// TIA Portal project "IndustrialSortingAutomation" (V17)
// Vorlageprojekt für das Buch mit Zielsystem S7-1200

(* hardware
DEVICE "S7-1200-Station_1"  S7-1200 Station
   slot 0: "Baugruppenträger_0"  Rack  V1.0
   slot 1: "PLC_1"  CPU 1211C DC/DC/DC  6ES7 211-1AE40-0XB0  V4.1
DEVICE "HMI_1"  KTP900 Basic PN
   slot 0: "HMI_1"  KTP900 Basic PN  6AV2 123-2JB03-0AX0  17.0.0.0
   slot 1: "HMI_RT_1"  KTP900 Basic PN  6AV2 123-2JB03-0AX0  17.0.0.0
   slot 5: "HMI_1.IE_CP_1"  PROFINET Interface  17.0.0.0
      slot 1: "PROFINET Interface_1"  PROFINET Interface
         slot 1: "Port_1"  Port
*)

// ===== PLC "PLC_1"  CPU 1211C DC/DC/DC =====

VAR_GLOBAL   // PLC tag table "Standard-Variablentabelle"
   "Motore_P" AT %A0.0 : Bool;
   "Sensore_P" AT %E0.0 : Bool;
   "Sensore_R" AT %E0.1 : Bool;
   "System_Byte" AT %MB1 : Byte;
   "FirstScan" AT %M1.0 : Bool;
   "DiagStatusUpdate" AT %M1.1 : Bool;
   "AlwaysTRUE" AT %M1.2 : Bool;
   "AlwaysFALSE" AT %M1.3 : Bool;
   "M_Pronto_P" AT %M10.0 : Bool;
   "M_Pronto_R" AT %M10.1 : Bool;
   "M_VAI_P" AT %M10.2 : Bool;
   "M_VAI_R" AT %M10.3 : Bool;
   "Cont_B_Board" AT %QW30 : Int;
   "Cont_V_Board" AT %QW32 : Int;
   "Cont_G_Board" AT %QW34 : Int;
   "Cont_P_Board" AT %QW36 : Int;
   "Motore_R" AT %Q0.1 : Bool;
   "Sorter_Pacchi_Turn" AT %Q0.2 : Bool;
   "Sorter_Pacchi_Belt" AT %Q0.3 : Bool;
   "Motore_Nastro_Ingresso_Smistamento" AT %Q0.4 : Bool;
   "Sorter_Raw_Blu_Turn" AT %Q0.5 : Bool;
   "Sorter_Raw_Blu_Belt" AT %Q0.6 : Bool;
   "Sorter_Raw_Verde_Turn" AT %Q0.7 : Bool;
   "Sorter_Raw_Verde_Belt" AT %Q1.0 : Bool;
   "Sorter_Raw_Grigio_Turn" AT %Q1.1 : Bool;
   "Sorter_Raw_Grigio_Belt" AT %Q1.2 : Bool;
   "Motore_Nastro_Comune" AT %Q2.0 : Bool;
   "Motore_Nastro_Uscita_P" AT %Q2.1 : Bool;
   "Motore_Nastro_Uscita_R" AT %Q2.2 : Bool;
   "Motore_Nastro_Smistamento" AT %Q2.3 : Bool;
   "Motore_Nastro_Uscita_B" AT %Q2.4 : Bool;
   "Motore_Nastro_Uscita_V" AT %Q2.5 : Bool;
   "Motore_Nastro_Uscita_G" AT %Q2.6 : Bool;
   "Sensore_Deviatore__P" AT %I0.2 : Bool;
   "Sensore_Uscita_P" AT %I0.3 : Bool;
   "Sensore_Uscita_R" AT %I0.4 : Bool;
   "Sensore_Fine_Incrocio" AT %I0.5 : Bool;
   "M_Apri_Grigio" AT %M2.2 : Bool;
   "M_AVA_Smistamento" AT %M2.3 : Bool;
   "M_Apri_Blu" AT %M2.0 : Bool;
   "M_Apri_Verde" AT %M2.1 : Bool;
   "Vision_Sensor" AT %IW30 : Int;
   "Cont_B" AT %MW100 : Int;
   "Cont_V" AT %MW102 : Int;
   "Cont_G" AT %MW104 : Int;
   "Cont_P" AT %MW106 : Int;
   "Emergency_Stop" AT %I0.6 : Bool;
   "Waring_Light" AT %Q1.3 : Bool;
   "M_Motore_P" AT %M3.0 : Bool;
   "M_Motore_R" AT %M3.1 : Bool;
   "M_Turn_P" AT %M3.2 : Bool;
   "M_Belt_P" AT %M3.3 : Bool;
   "M_Turn_B" AT %M3.4 : Bool;
   "M_Belt_B" AT %M3.5 : Bool;
   "M_Turn_V" AT %M3.6 : Bool;
   "M_Belt_V" AT %M3.7 : Bool;
   "M_Turn_G" AT %M4.0 : Bool;
   "M_Belt_G" AT %M4.1 : Bool;
   "Alarm_Siren" AT %Q1.4 : Bool;
END_VAR

DATA_BLOCK "FB_Nastro_Ingresso_DB_Pacchi"   // DB1
{ S7_Optimized_Access := 'TRUE' }
VERSION : 0.1
// stored: InstanceOfName FB_Nastro_Ingresso
"FB_Nastro_Ingresso"
BEGIN
END_DATA_BLOCK

DATA_BLOCK "FB_Nastro_Ingresso_DB_Raw"   // DB2
{ S7_Optimized_Access := 'TRUE' }
VERSION : 0.1
// stored: InstanceOfName FB_Nastro_Ingresso
"FB_Nastro_Ingresso"
BEGIN
END_DATA_BLOCK

DATA_BLOCK "FB_Gestore_Incrocio_DB"   // DB3
{ S7_Optimized_Access := 'TRUE' }
VERSION : 0.1
// stored: InstanceOfName FB_Gestore_Incrocio
"FB_Gestore_Incrocio"
BEGIN
END_DATA_BLOCK

DATA_BLOCK "FB_Deviatore_DB_Pacchi"   // DB4
{ S7_Optimized_Access := 'TRUE' }
VERSION : 0.1
// stored: InstanceOfName FB_Deviatore
"FB_Deviatore"
BEGIN
END_DATA_BLOCK

DATA_BLOCK "FB_Gestore_Smistamento_DB"   // DB5
{ S7_Optimized_Access := 'TRUE' }
VERSION : 0.1
// stored: InstanceOfName FB_Gestore_Smistamento
"FB_Gestore_Smistamento"
BEGIN
END_DATA_BLOCK

DATA_BLOCK "FB_Deviatore_DB_Blu"   // DB6
{ S7_Optimized_Access := 'TRUE' }
VERSION : 0.1
// stored: InstanceOfName FB_Deviatore
"FB_Deviatore"
BEGIN
END_DATA_BLOCK

DATA_BLOCK "FB_Deviatore_DB_Verde"   // DB7
{ S7_Optimized_Access := 'TRUE' }
VERSION : 0.1
// stored: InstanceOfName FB_Deviatore
"FB_Deviatore"
BEGIN
END_DATA_BLOCK

DATA_BLOCK "FB_Deviatore_DB_Grigio"   // DB8
{ S7_Optimized_Access := 'TRUE' }
VERSION : 0.1
// stored: InstanceOfName FB_Deviatore
"FB_Deviatore"
BEGIN
END_DATA_BLOCK

// folder: System blocks/Program resources

DATA_BLOCK "IEC_Timer_0_DB_Nastro_Smistamento"   // DB9
{ S7_Optimized_Access := 'TRUE' }
AUTHOR : Simatic
FAMILY : IEC
NAME : IEC_TMR
VERSION : 1.0
// stored: InstanceOfName IEC_TIMER
"IEC_TIMER"
BEGIN
END_DATA_BLOCK

// folder: (top level)

FUNCTION_BLOCK "FB_Nastro_Ingresso"   // FB1, LAD
{ S7_Optimized_Access := 'TRUE' }
VERSION : 0.1
   VAR_INPUT
      fn : Bool;
      VAI : Bool;
      Tempo_Spinta : Time;
   END_VAR
   VAR_OUTPUT
      AVA : Bool;
      pronto : Bool;
   END_VAR
   VAR
      f0 : Bool;
      f1 : Bool;
      f2 : Bool;
      f3 : Bool;
      tr1 : Bool;
      tr2 : Bool;
      tr3 : Bool;
      tr4 : Bool;
      Timer_Attr : IEC_TIMER;
   END_VAR
BEGIN

REGION Network 1: Inizializzazione
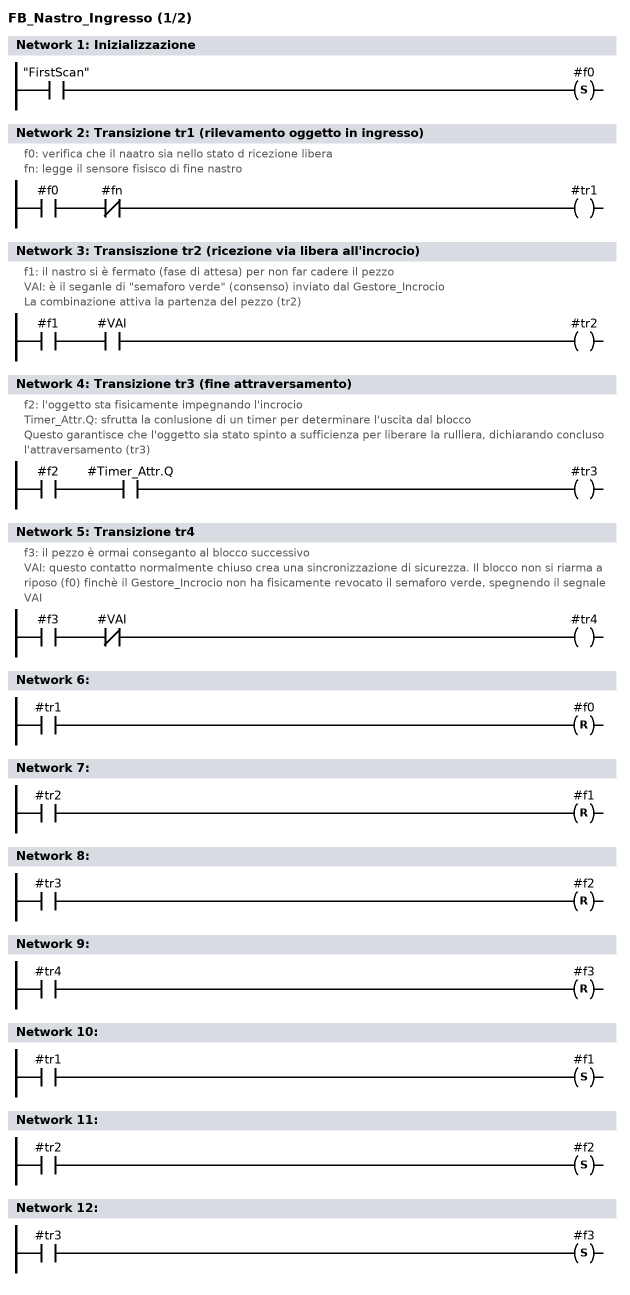
   RUNG wire#powerrail
      Contact( "FirstScan" )
      S_Coil( #f0 )
   END_RUNG
   // the same network as SCL:
   IF "FirstScan" THEN #f0 := TRUE; END_IF;
END_REGION

REGION Network 2: Transizione tr1 (rilevamento oggetto in ingresso)
   // f0: verifica che il naatro sia nello stato d ricezione libera
   // fn: legge il sensore fisisco di fine nastro
   RUNG wire#powerrail
      Contact( #f0 )
      I_Contact( #fn )
      Coil( #tr1 )
   END_RUNG
   // the same network as SCL:
   #tr1 := #f0 AND NOT #fn;
END_REGION

REGION Network 3: Transiszione tr2 (ricezione via libera all'incrocio)
   // f1: il nastro si è fermato (fase di attesa) per non far cadere il pezzo
   // VAI: è il seganle di "semaforo verde" (consenso) inviato dal Gestore_Incrocio
   // La combinazione attiva la partenza del pezzo (tr2)
   RUNG wire#powerrail
      Contact( #f1 )
      Contact( #VAI )
      Coil( #tr2 )
   END_RUNG
   // the same network as SCL:
   #tr2 := #f1 AND #VAI;
END_REGION

REGION Network 4: Transizione tr3 (fine attraversamento)
   // f2: l'oggetto sta fisicamente impegnando l'incrocio
   // Timer_Attr.Q: sfrutta la conlusione di un timer per determinare l'uscita dal blocco
   // Questo garantisce che l'oggetto sia stato spinto a sufficienza per liberare la rulliera, dichiarando concluso l'attraversamento (tr3)
   RUNG wire#powerrail
      Contact( #f2 )
      Contact( #Timer_Attr.Q )
      Coil( #tr3 )
   END_RUNG
   // the same network as SCL:
   #tr3 := #f2 AND #Timer_Attr.Q;
END_REGION

REGION Network 5: Transizione tr4
   // f3: il pezzo è ormai conseganto al blocco successivo 
   // VAI: questo contatto normalmente chiuso crea una sincronizzazione di sicurezza. Il blocco non si riarma a riposo (f0) finchè il Gestore_Incrocio non ha fisicamente revocato il semaforo verde, spegnendo il segnale VAI
   RUNG wire#powerrail
      Contact( #f3 )
      I_Contact( #VAI )
      Coil( #tr4 )
   END_RUNG
   // the same network as SCL:
   #tr4 := #f3 AND NOT #VAI;
END_REGION

REGION Network 6
   RUNG wire#powerrail
      Contact( #tr1 )
      R_Coil( #f0 )
   END_RUNG
   // the same network as SCL:
   IF #tr1 THEN #f0 := FALSE; END_IF;
END_REGION

REGION Network 7
   RUNG wire#powerrail
      Contact( #tr2 )
      R_Coil( #f1 )
   END_RUNG
   // the same network as SCL:
   IF #tr2 THEN #f1 := FALSE; END_IF;
END_REGION

REGION Network 8
   RUNG wire#powerrail
      Contact( #tr3 )
      R_Coil( #f2 )
   END_RUNG
   // the same network as SCL:
   IF #tr3 THEN #f2 := FALSE; END_IF;
END_REGION

REGION Network 9
   RUNG wire#powerrail
      Contact( #tr4 )
      R_Coil( #f3 )
   END_RUNG
   // the same network as SCL:
   IF #tr4 THEN #f3 := FALSE; END_IF;
END_REGION

REGION Network 10
   RUNG wire#powerrail
      Contact( #tr1 )
      S_Coil( #f1 )
   END_RUNG
   // the same network as SCL:
   IF #tr1 THEN #f1 := TRUE; END_IF;
END_REGION

REGION Network 11
   RUNG wire#powerrail
      Contact( #tr2 )
      S_Coil( #f2 )
   END_RUNG
   // the same network as SCL:
   IF #tr2 THEN #f2 := TRUE; END_IF;
END_REGION

REGION Network 12
   RUNG wire#powerrail
      Contact( #tr3 )
      S_Coil( #f3 )
   END_RUNG
   // the same network as SCL:
   IF #tr3 THEN #f3 := TRUE; END_IF;
END_REGION

REGION Network 13
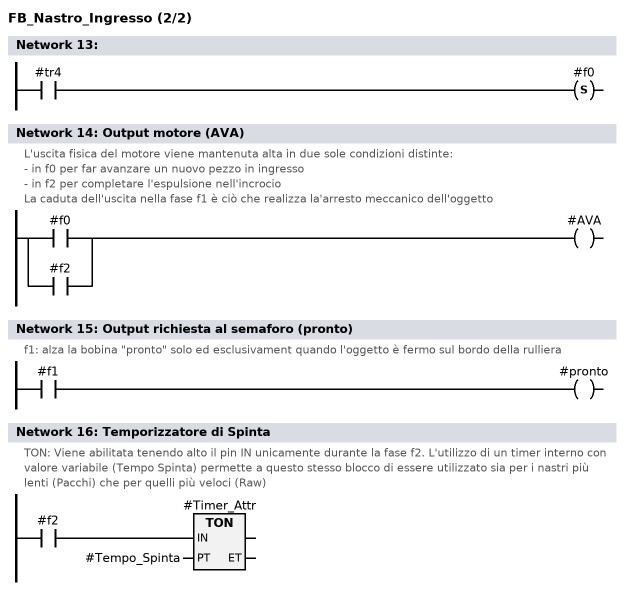
   RUNG wire#powerrail
      Contact( #tr4 )
      S_Coil( #f0 )
   END_RUNG
   // the same network as SCL:
   IF #tr4 THEN #f0 := TRUE; END_IF;
END_REGION

REGION Network 14: Output motore (AVA)
   // L'uscita fisica del motore viene mantenuta alta in due sole condizioni distinte:
   // - in f0 per far avanzare un nuovo pezzo in ingresso
   // - in f2 per completare l'espulsione nell'incrocio
   // La caduta dell'uscita nella fase f1 è ciò che realizza la'arresto meccanico dell'oggetto
   RUNG wire#powerrail
      Contact( #f0 )
      wire#w1
      Coil( #AVA )
   END_RUNG
   RUNG wire#powerrail
      Contact( #f2 )
   END_RUNG wire#w1
   // the same network as SCL:
   #AVA := #f0 OR #f2;
END_REGION

REGION Network 15: Output richiesta al semaforo (pronto)
   // f1: alza la bobina "pronto" solo ed esclusivament quando l'oggetto è fermo sul bordo della rulliera
   RUNG wire#powerrail
      Contact( #f1 )
      Coil( #pronto )
   END_RUNG
   // the same network as SCL:
   #pronto := #f1;
END_REGION

REGION Network 16: Temporizzatore di Spinta
   // TON: Viene abilitata tenendo alto il pin IN unicamente durante la fase f2. L'utilizzo di un timer interno con valore variabile (Tempo Spinta) permette a questo stesso blocco di essere utilizzato sia per i nastri più lenti (Pacchi) che per quelli più veloci (Raw)
   #Timer_Attr.TON(IN := #f2, PT := #Tempo_Spinta);
END_REGION
END_FUNCTION_BLOCK

FUNCTION_BLOCK "FB_Gestore_Incrocio"   // FB2, LAD
{ S7_Optimized_Access := 'TRUE' }
VERSION : 0.1
   VAR_INPUT
      pronto_P : Bool;
      pronto_R : Bool;
      Pass : Bool;
   END_VAR
   VAR_OUTPUT
      VAI_P : Bool;
      VAI_R : Bool;
   END_VAR
   VAR
      f0 : Bool;
      f1 : Bool;
      f2 : Bool;
      tr1 : Bool;
      tr2 : Bool;
      tr3 : Bool;
      tr4 : Bool;
      Mem_Fronte_P : Bool;
      Mem_Fronte_R : Bool;
   END_VAR
   VAR_TEMP   // added for the SCL form of the ladder/FBD networks
      _w1 : Bool;
   END_VAR
BEGIN

REGION Network 1: Inizializzazione
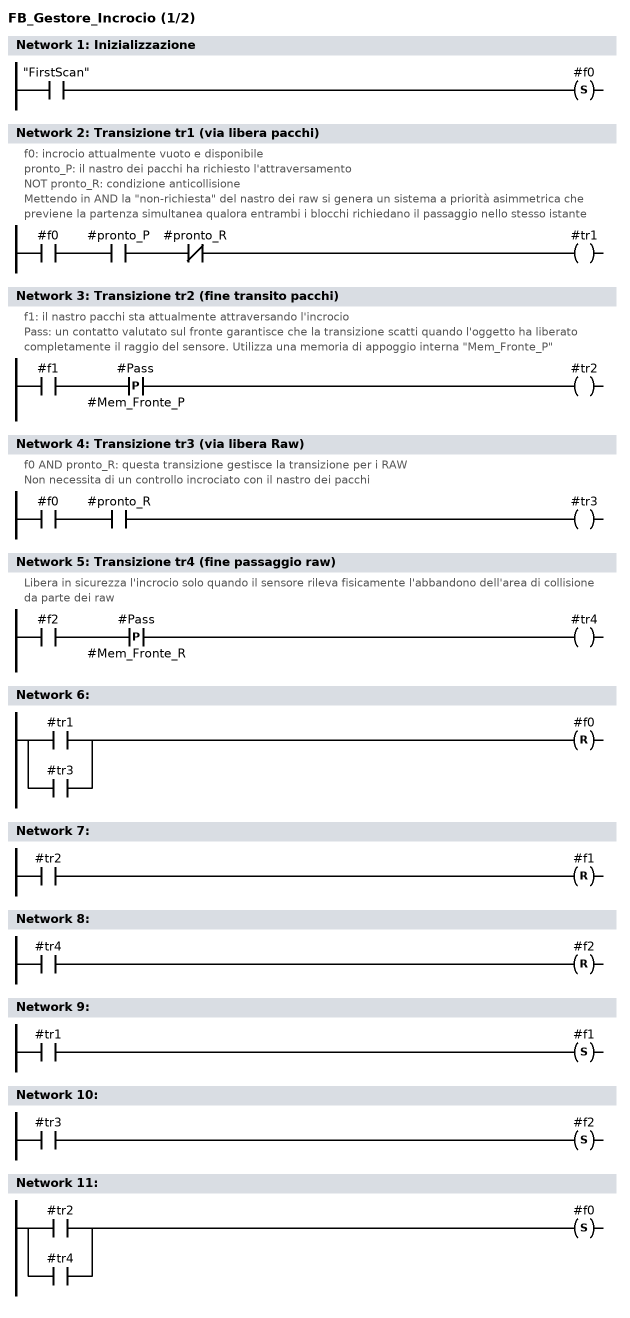
   RUNG wire#powerrail
      Contact( "FirstScan" )
      S_Coil( #f0 )
   END_RUNG
   // the same network as SCL:
   IF "FirstScan" THEN #f0 := TRUE; END_IF;
END_REGION

REGION Network 2: Transizione tr1 (via libera pacchi)
   // f0: incrocio attualmente vuoto e disponibile
   // pronto_P: il nastro dei pacchi ha richiesto l'attraversamento
   // NOT pronto_R: condizione anticollisione
   // Mettendo in AND la "non-richiesta" del nastro dei raw si genera un sistema a priorità asimmetrica che previene la partenza simultanea qualora entrambi i blocchi richiedano il passaggio nello stesso istante
   RUNG wire#powerrail
      Contact( #f0 )
      Contact( #pronto_P )
      I_Contact( #pronto_R )
      Coil( #tr1 )
   END_RUNG
   // the same network as SCL:
   #tr1 := #f0 AND #pronto_P AND NOT #pronto_R;
END_REGION

REGION Network 3: Transizione tr2 (fine transito pacchi)
   // f1: il nastro pacchi sta attualmente attraversando l'incrocio
   // Pass: un contatto valutato sul fronte garantisce che la transizione scatti quando l'oggetto ha liberato completamente il raggio del sensore. Utilizza una memoria di appoggio interna "Mem_Fronte_P"
   RUNG wire#powerrail
      Contact( #f1 )
      P_Contact(operand := #Pass, bit := #Mem_Fronte_P)
      Coil( #tr2 )
   END_RUNG
   // the same network as SCL:
   #_w1 := #f1 AND #Pass AND NOT #Mem_Fronte_P;   // rising edge of #Pass
   #Mem_Fronte_P := #Pass;
   #tr2 := #_w1;
END_REGION

REGION Network 4: Transizione tr3 (via libera Raw)
   // f0 AND pronto_R: questa transizione gestisce la transizione per i RAW
   // Non necessita di un controllo incrociato con il nastro dei pacchi
   RUNG wire#powerrail
      Contact( #f0 )
      Contact( #pronto_R )
      Coil( #tr3 )
   END_RUNG
   // the same network as SCL:
   #tr3 := #f0 AND #pronto_R;
END_REGION

REGION Network 5: Transizione tr4 (fine passaggio raw)
   // Libera in sicurezza l'incrocio solo quando il sensore rileva fisicamente l'abbandono dell'area di collisione da parte dei raw
   RUNG wire#powerrail
      Contact( #f2 )
      P_Contact(operand := #Pass, bit := #Mem_Fronte_R)
      Coil( #tr4 )
   END_RUNG
   // the same network as SCL:
   #_w1 := #f2 AND #Pass AND NOT #Mem_Fronte_R;   // rising edge of #Pass
   #Mem_Fronte_R := #Pass;
   #tr4 := #_w1;
END_REGION

REGION Network 6
   RUNG wire#powerrail
      Contact( #tr1 )
      wire#w1
      R_Coil( #f0 )
   END_RUNG
   RUNG wire#powerrail
      Contact( #tr3 )
   END_RUNG wire#w1
   // the same network as SCL:
   IF #tr1 OR #tr3 THEN #f0 := FALSE; END_IF;
END_REGION

REGION Network 7
   RUNG wire#powerrail
      Contact( #tr2 )
      R_Coil( #f1 )
   END_RUNG
   // the same network as SCL:
   IF #tr2 THEN #f1 := FALSE; END_IF;
END_REGION

REGION Network 8
   RUNG wire#powerrail
      Contact( #tr4 )
      R_Coil( #f2 )
   END_RUNG
   // the same network as SCL:
   IF #tr4 THEN #f2 := FALSE; END_IF;
END_REGION

REGION Network 9
   RUNG wire#powerrail
      Contact( #tr1 )
      S_Coil( #f1 )
   END_RUNG
   // the same network as SCL:
   IF #tr1 THEN #f1 := TRUE; END_IF;
END_REGION

REGION Network 10
   RUNG wire#powerrail
      Contact( #tr3 )
      S_Coil( #f2 )
   END_RUNG
   // the same network as SCL:
   IF #tr3 THEN #f2 := TRUE; END_IF;
END_REGION

REGION Network 11
   RUNG wire#powerrail
      Contact( #tr2 )
      wire#w1
      S_Coil( #f0 )
   END_RUNG
   RUNG wire#powerrail
      Contact( #tr4 )
   END_RUNG wire#w1
   // the same network as SCL:
   IF #tr2 OR #tr4 THEN #f0 := TRUE; END_IF;
END_REGION

REGION Network 12: Output consenso pacchi
   // VAI_P: il segnale di "semaforo verde" per la linea dei pacchi  viene pilotato dallo stato f1. Finchè f1 è ativo il permesso rimane alto generando il flusso continuo.
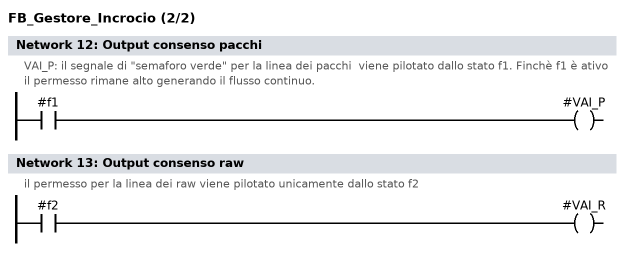
   RUNG wire#powerrail
      Contact( #f1 )
      Coil( #VAI_P )
   END_RUNG
   // the same network as SCL:
   #VAI_P := #f1;
END_REGION

REGION Network 13: Output consenso raw
   // il permesso per la linea dei raw viene pilotato unicamente dallo stato f2
   RUNG wire#powerrail
      Contact( #f2 )
      Coil( #VAI_R )
   END_RUNG
   // the same network as SCL:
   #VAI_R := #f2;
END_REGION
END_FUNCTION_BLOCK

FUNCTION_BLOCK "FB_Deviatore"   // FB3, LAD
{ S7_Optimized_Access := 'TRUE' }
VERSION : 0.1
   VAR_INPUT
      Apri : Bool;
      Pass : Bool;
   END_VAR
   VAR_OUTPUT
      Ruota : Bool;
      Nastro_Pivot : Bool;
   END_VAR
   VAR
      f0 : Bool;
      f1 : Bool;
      tr1 : Bool;
      tr2 : Bool;
   END_VAR
BEGIN

REGION Network 1: Inizializzazione
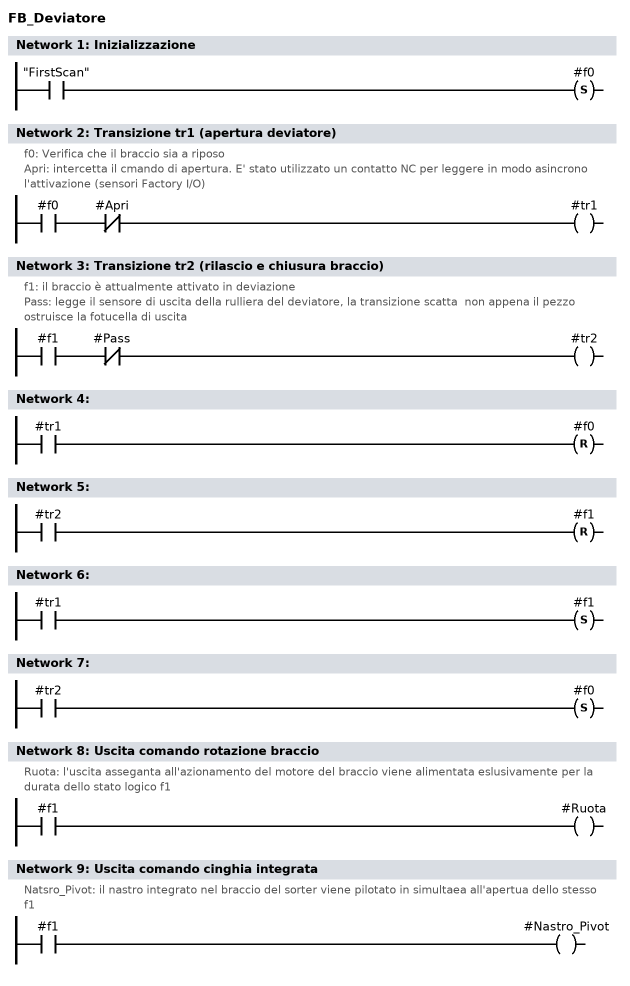
   RUNG wire#powerrail
      Contact( "FirstScan" )
      S_Coil( #f0 )
   END_RUNG
   // the same network as SCL:
   IF "FirstScan" THEN #f0 := TRUE; END_IF;
END_REGION

REGION Network 2: Transizione tr1 (apertura deviatore)
   // f0: Verifica che il braccio sia a riposo
   // Apri: intercetta il cmando di apertura. E' stato utilizzato un contatto NC per leggere in modo asincrono l'attivazione (sensori Factory I/O)
   RUNG wire#powerrail
      Contact( #f0 )
      I_Contact( #Apri )
      Coil( #tr1 )
   END_RUNG
   // the same network as SCL:
   #tr1 := #f0 AND NOT #Apri;
END_REGION

REGION Network 3: Transizione tr2 (rilascio e chiusura braccio)
   // f1: il braccio è attualmente attivato in deviazione
   // Pass: legge il sensore di uscita della rulliera del deviatore, la transizione scatta  non appena il pezzo ostruisce la fotucella di uscita
   RUNG wire#powerrail
      Contact( #f1 )
      I_Contact( #Pass )
      Coil( #tr2 )
   END_RUNG
   // the same network as SCL:
   #tr2 := #f1 AND NOT #Pass;
END_REGION

REGION Network 4
   RUNG wire#powerrail
      Contact( #tr1 )
      R_Coil( #f0 )
   END_RUNG
   // the same network as SCL:
   IF #tr1 THEN #f0 := FALSE; END_IF;
END_REGION

REGION Network 5
   RUNG wire#powerrail
      Contact( #tr2 )
      R_Coil( #f1 )
   END_RUNG
   // the same network as SCL:
   IF #tr2 THEN #f1 := FALSE; END_IF;
END_REGION

REGION Network 6
   RUNG wire#powerrail
      Contact( #tr1 )
      S_Coil( #f1 )
   END_RUNG
   // the same network as SCL:
   IF #tr1 THEN #f1 := TRUE; END_IF;
END_REGION

REGION Network 7
   RUNG wire#powerrail
      Contact( #tr2 )
      S_Coil( #f0 )
   END_RUNG
   // the same network as SCL:
   IF #tr2 THEN #f0 := TRUE; END_IF;
END_REGION

REGION Network 8: Uscita comando rotazione braccio
   // Ruota: l'uscita asseganta all'azionamento del motore del braccio viene alimentata eslusivamente per la durata dello stato logico f1
   RUNG wire#powerrail
      Contact( #f1 )
      Coil( #Ruota )
   END_RUNG
   // the same network as SCL:
   #Ruota := #f1;
END_REGION

REGION Network 9: Uscita comando cinghia integrata
   // Natsro_Pivot: il nastro integrato nel braccio del sorter viene pilotato in simultaea all'apertua dello stesso f1
   RUNG wire#powerrail
      Contact( #f1 )
      Coil( #Nastro_Pivot )
   END_RUNG
   // the same network as SCL:
   #Nastro_Pivot := #f1;
END_REGION
END_FUNCTION_BLOCK

FUNCTION_BLOCK "FB_Gestore_Smistamento"   // FB4, LAD
{ S7_Optimized_Access := 'TRUE' }
VERSION : 0.1
   VAR_INPUT
      Vis_C : Int;   // Vision sensor per i colori
      Pass : Bool;
   END_VAR
   VAR_OUTPUT
      AVA : Bool;
      Apri_B : Bool;
      Apri_V : Bool;
      Apri_G : Bool;
   END_VAR
   VAR
      f0 : Bool;
      f1 : Bool;
      f2 : Bool;
      f3 : Bool;
      tr1 : Bool;
      tr2 : Bool;
      tr3 : Bool;
      tr4 : Bool;
      tr5 : Bool;
      tr6 : Bool;
   END_VAR
BEGIN

REGION Network 1: Inizializzazione
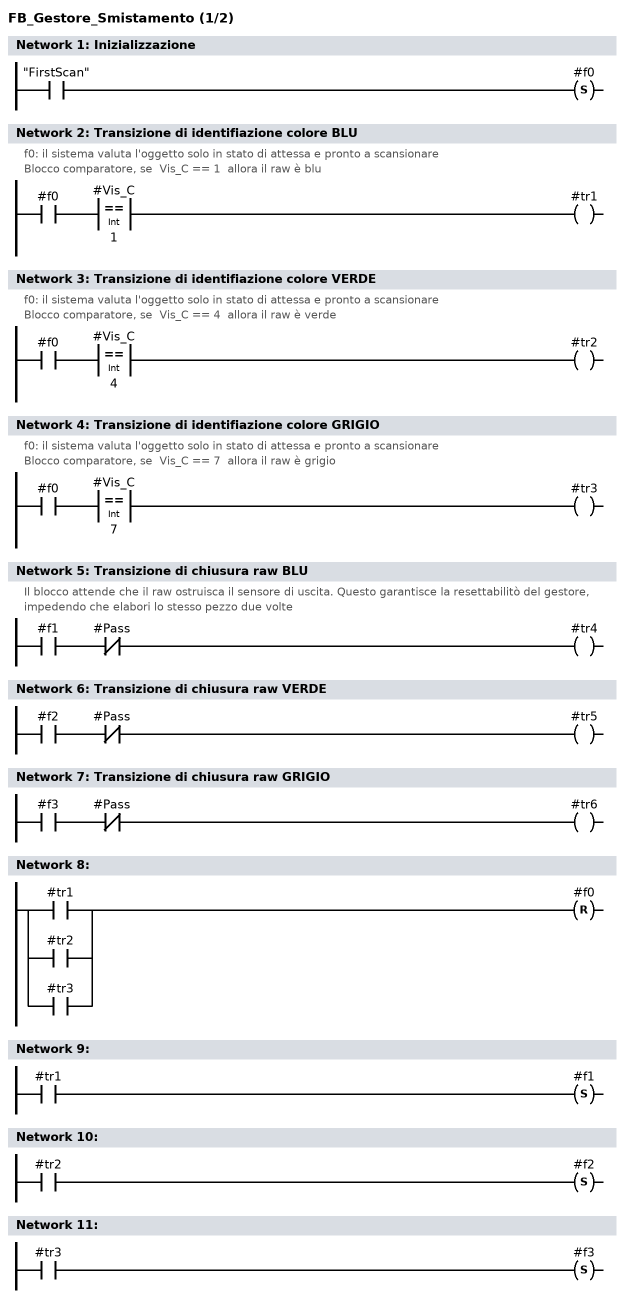
   RUNG wire#powerrail
      Contact( "FirstScan" )
      S_Coil( #f0 )
   END_RUNG
   // the same network as SCL:
   IF "FirstScan" THEN #f0 := TRUE; END_IF;
END_REGION

REGION Network 2: Transizione di identifiazione colore BLU
   // f0: il sistema valuta l'oggetto solo in stato di attessa e pronto a scansionare
   // Blocco comparatore, se  Vis_C == 1  allora il raw è blu
   RUNG wire#powerrail
      Contact( #f0 )
      { S7_Templates := "SrcType := Int" } EQ_Contact(in1 := #Vis_C, in2 := 1)
      Coil( #tr1 )
   END_RUNG
   // the same network as SCL:
   #tr1 := #f0 AND (#Vis_C = 1);
END_REGION

REGION Network 3: Transizione di identifiazione colore VERDE
   // f0: il sistema valuta l'oggetto solo in stato di attessa e pronto a scansionare
   // Blocco comparatore, se  Vis_C == 4  allora il raw è verde
   RUNG wire#powerrail
      Contact( #f0 )
      { S7_Templates := "SrcType := Int" } EQ_Contact(in1 := #Vis_C, in2 := 4)
      Coil( #tr2 )
   END_RUNG
   // the same network as SCL:
   #tr2 := #f0 AND (#Vis_C = 4);
END_REGION

REGION Network 4: Transizione di identifiazione colore GRIGIO
   // f0: il sistema valuta l'oggetto solo in stato di attessa e pronto a scansionare
   // Blocco comparatore, se  Vis_C == 7  allora il raw è grigio
   RUNG wire#powerrail
      Contact( #f0 )
      { S7_Templates := "SrcType := Int" } EQ_Contact(in1 := #Vis_C, in2 := 7)
      Coil( #tr3 )
   END_RUNG
   // the same network as SCL:
   #tr3 := #f0 AND (#Vis_C = 7);
END_REGION

REGION Network 5: Transizione di chiusura raw BLU
   // Il blocco attende che il raw ostruisca il sensore di uscita. Questo garantisce la resettabilitò del gestore, impedendo che elabori lo stesso pezzo due volte
   RUNG wire#powerrail
      Contact( #f1 )
      I_Contact( #Pass )
      Coil( #tr4 )
   END_RUNG
   // the same network as SCL:
   #tr4 := #f1 AND NOT #Pass;
END_REGION

REGION Network 6: Transizione di chiusura raw VERDE
   RUNG wire#powerrail
      Contact( #f2 )
      I_Contact( #Pass )
      Coil( #tr5 )
   END_RUNG
   // the same network as SCL:
   #tr5 := #f2 AND NOT #Pass;
END_REGION

REGION Network 7: Transizione di chiusura raw GRIGIO
   RUNG wire#powerrail
      Contact( #f3 )
      I_Contact( #Pass )
      Coil( #tr6 )
   END_RUNG
   // the same network as SCL:
   #tr6 := #f3 AND NOT #Pass;
END_REGION

REGION Network 8
   RUNG wire#powerrail
      Contact( #tr1 )
      wire#w1
      R_Coil( #f0 )
   END_RUNG
   RUNG wire#powerrail
      Contact( #tr2 )
   END_RUNG wire#w1
   RUNG wire#powerrail
      Contact( #tr3 )
   END_RUNG wire#w1
   // the same network as SCL:
   IF #tr1 OR #tr2 OR #tr3 THEN #f0 := FALSE; END_IF;
END_REGION

REGION Network 9
   RUNG wire#powerrail
      Contact( #tr1 )
      S_Coil( #f1 )
   END_RUNG
   // the same network as SCL:
   IF #tr1 THEN #f1 := TRUE; END_IF;
END_REGION

REGION Network 10
   RUNG wire#powerrail
      Contact( #tr2 )
      S_Coil( #f2 )
   END_RUNG
   // the same network as SCL:
   IF #tr2 THEN #f2 := TRUE; END_IF;
END_REGION

REGION Network 11
   RUNG wire#powerrail
      Contact( #tr3 )
      S_Coil( #f3 )
   END_RUNG
   // the same network as SCL:
   IF #tr3 THEN #f3 := TRUE; END_IF;
END_REGION

REGION Network 12
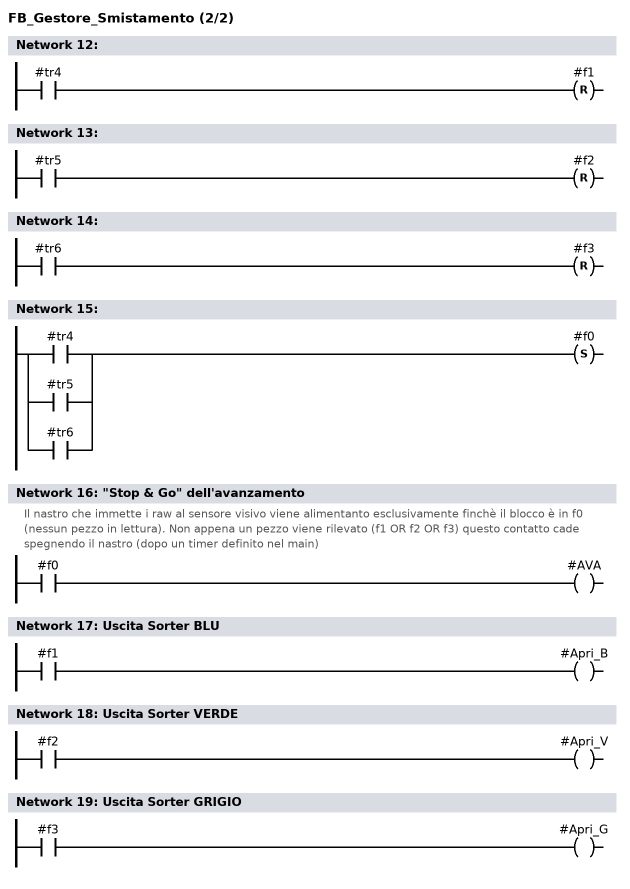
   RUNG wire#powerrail
      Contact( #tr4 )
      R_Coil( #f1 )
   END_RUNG
   // the same network as SCL:
   IF #tr4 THEN #f1 := FALSE; END_IF;
END_REGION

REGION Network 13
   RUNG wire#powerrail
      Contact( #tr5 )
      R_Coil( #f2 )
   END_RUNG
   // the same network as SCL:
   IF #tr5 THEN #f2 := FALSE; END_IF;
END_REGION

REGION Network 14
   RUNG wire#powerrail
      Contact( #tr6 )
      R_Coil( #f3 )
   END_RUNG
   // the same network as SCL:
   IF #tr6 THEN #f3 := FALSE; END_IF;
END_REGION

REGION Network 15
   RUNG wire#powerrail
      Contact( #tr4 )
      wire#w1
      S_Coil( #f0 )
   END_RUNG
   RUNG wire#powerrail
      Contact( #tr5 )
   END_RUNG wire#w1
   RUNG wire#powerrail
      Contact( #tr6 )
   END_RUNG wire#w1
   // the same network as SCL:
   IF #tr4 OR #tr5 OR #tr6 THEN #f0 := TRUE; END_IF;
END_REGION

REGION Network 16: "Stop & Go" dell'avanzamento
   // Il nastro che immette i raw al sensore visivo viene alimentanto esclusivamente finchè il blocco è in f0 (nessun pezzo in lettura). Non appena un pezzo viene rilevato (f1 OR f2 OR f3) questo contatto cade spegnendo il nastro (dopo un timer definito nel main)
   RUNG wire#powerrail
      Contact( #f0 )
      Coil( #AVA )
   END_RUNG
   // the same network as SCL:
   #AVA := #f0;
END_REGION

REGION Network 17: Uscita Sorter BLU
   RUNG wire#powerrail
      Contact( #f1 )
      Coil( #Apri_B )
   END_RUNG
   // the same network as SCL:
   #Apri_B := #f1;
END_REGION

REGION Network 18: Uscita Sorter VERDE
   RUNG wire#powerrail
      Contact( #f2 )
      Coil( #Apri_V )
   END_RUNG
   // the same network as SCL:
   #Apri_V := #f2;
END_REGION

REGION Network 19: Uscita Sorter GRIGIO
   RUNG wire#powerrail
      Contact( #f3 )
      Coil( #Apri_G )
   END_RUNG
   // the same network as SCL:
   #Apri_G := #f3;
END_REGION
END_FUNCTION_BLOCK

FUNCTION "MHJ-PLC-Lab-Function-S71200" : Void   // FC9000, SCL
{ S7_Optimized_Access := 'TRUE' }
VERSION : 0.1
   VAR_TEMP
      rdTimeReturn : Int;
      outputTime : DTL;
      SyncVal : Byte;
      forVal : Int;
      forVal_2 : Int;
      Value : Byte;
   END_VAR
   VAR CONSTANT
      CompVal : Byte := 16#34;
      Value_01 : Byte := 16#11;
      Value_01_DW : DWord := 16#A165_D992;
      Value_02_DW : DWord := 16#58BE_4401;
   END_VAR
BEGIN

   #Value:=PEEK(area := 16#82,
        dbNumber := 0,
        byteOffset := 511);
   #Value := #Value + 1;

   POKE(area := 16#82,
        dbNumber := 0,
        byteOffset := 511,
        value := #Value);

   POKE(area:=16#81,
        dbNumber:=0,
        byteOffset:=1016,
        value:=#Value_01_DW);
   POKE(area := 16#81,
        dbNumber := 0,
        byteOffset := 1020,
        value := #Value_02_DW);

   POKE(area := 16#81,
        dbNumber := 0,
        byteOffset := 511,
        value := B#16#00);

   FOR #forVal := 0 TO 120 DO
       FOR #forVal_2:=0 TO 10 DO
           #rdTimeReturn:=RD_SYS_T(#outputTime);
           #rdTimeReturn := WR_SYS_T(#outputTime);
           #rdTimeReturn := RD_SYS_T(#outputTime);
           #rdTimeReturn := WR_SYS_T(#outputTime);
       END_FOR;
       #SyncVal:= PEEK(area := 16#81,
                      dbNumber := 0,
                      byteOffset := 511);
       IF #SyncVal = #CompVal THEN
          GOTO M_1;
       END_IF;
   END_FOR;
   RETURN;

   M_1:
   POKE(area := 16#81,
        dbNumber := 0,
        byteOffset := 511,
        value := B#16#0);
END_FUNCTION

ORGANIZATION_BLOCK "Main"   // OB1, LAD, ProgramCycle
TITLE = "Main Program Sweep (Cycle)"
{ S7_Optimized_Access := 'TRUE' }
VERSION : 0.1
   VAR_INPUT
      Initial_Call : Bool;   // Initial call of this OB
      Remanence : Bool;   // =True, if remanent data are available
   END_VAR
BEGIN

REGION Network 1: Konnektierungsbaustein für PLC-Lab
   // Im Netzwerk 1 wird der Konnektierungsbaustein für PLC-Lab aufgerufen.
   // Dieser Aufruf darf nicht entfernt werden!
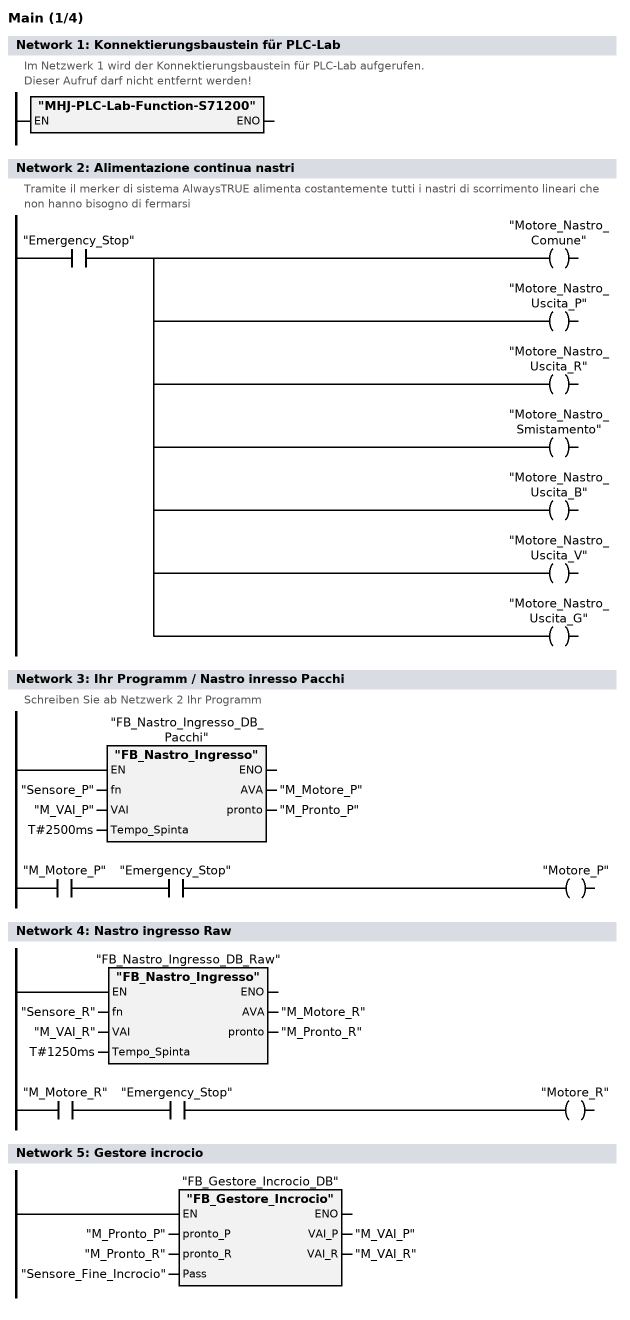
   RUNG wire#powerrail
      "MHJ-PLC-Lab-Function-S71200"()
   END_RUNG
   // the same network as SCL:
   "MHJ-PLC-Lab-Function-S71200"();
END_REGION

REGION Network 2: Alimentazione continua nastri
   // Tramite il merker di sistema AlwaysTRUE alimenta costantemente tutti i nastri di scorrimento lineari che non hanno bisogno di fermarsi
   RUNG wire#powerrail
      Contact( "Emergency_Stop" )
      wire#w1
      Coil( "Motore_Nastro_Comune" )
   END_RUNG
   RUNG wire#w1
      Coil( "Motore_Nastro_Uscita_P" )
   END_RUNG
   RUNG wire#w1
      Coil( "Motore_Nastro_Uscita_R" )
   END_RUNG
   RUNG wire#w1
      Coil( "Motore_Nastro_Smistamento" )
   END_RUNG
   RUNG wire#w1
      Coil( "Motore_Nastro_Uscita_B" )
   END_RUNG
   RUNG wire#w1
      Coil( "Motore_Nastro_Uscita_V" )
   END_RUNG
   RUNG wire#w1
      Coil( "Motore_Nastro_Uscita_G" )
   END_RUNG
   // the same network as SCL:
   "Motore_Nastro_Comune" := "Emergency_Stop";
   "Motore_Nastro_Uscita_P" := "Emergency_Stop";
   "Motore_Nastro_Uscita_R" := "Emergency_Stop";
   "Motore_Nastro_Smistamento" := "Emergency_Stop";
   "Motore_Nastro_Uscita_B" := "Emergency_Stop";
   "Motore_Nastro_Uscita_V" := "Emergency_Stop";
   "Motore_Nastro_Uscita_G" := "Emergency_Stop";
END_REGION

REGION Network 3: Ihr Programm / Nastro inresso Pacchi
   // Schreiben Sie ab Netzwerk 2 Ihr Programm
   RUNG wire#powerrail
      "FB_Nastro_Ingresso_DB_Pacchi"(fn := "Sensore_P", VAI := "M_VAI_P", Tempo_Spinta := T#2500ms, AVA => "M_Motore_P", pronto => "M_Pronto_P")
   END_RUNG
   RUNG wire#powerrail
      Contact( "M_Motore_P" )
      Contact( "Emergency_Stop" )
      Coil( "Motore_P" )
   END_RUNG
   // the same network as SCL:
   "FB_Nastro_Ingresso_DB_Pacchi"(fn := "Sensore_P",   // "FB_Nastro_Ingresso"
                           VAI := "M_VAI_P",
                           Tempo_Spinta := T#2500ms,
                           AVA => "M_Motore_P",
                           pronto => "M_Pronto_P");
   "Motore_P" := "M_Motore_P" AND "Emergency_Stop";
END_REGION

REGION Network 4: Nastro ingresso Raw
   RUNG wire#powerrail
      "FB_Nastro_Ingresso_DB_Raw"(fn := "Sensore_R", VAI := "M_VAI_R", Tempo_Spinta := T#1250ms, AVA => "M_Motore_R", pronto => "M_Pronto_R")
   END_RUNG
   RUNG wire#powerrail
      Contact( "M_Motore_R" )
      Contact( "Emergency_Stop" )
      Coil( "Motore_R" )
   END_RUNG
   // the same network as SCL:
   "FB_Nastro_Ingresso_DB_Raw"(fn := "Sensore_R",   // "FB_Nastro_Ingresso"
                           VAI := "M_VAI_R",
                           Tempo_Spinta := T#1250ms,
                           AVA => "M_Motore_R",
                           pronto => "M_Pronto_R");
   "Motore_R" := "M_Motore_R" AND "Emergency_Stop";
END_REGION

REGION Network 5: Gestore incrocio
   RUNG wire#powerrail
      "FB_Gestore_Incrocio_DB"(pronto_P := "M_Pronto_P", pronto_R := "M_Pronto_R", Pass := "Sensore_Fine_Incrocio", VAI_P => "M_VAI_P", VAI_R => "M_VAI_R")
   END_RUNG
   // the same network as SCL:
   "FB_Gestore_Incrocio_DB"(pronto_P := "M_Pronto_P",   // "FB_Gestore_Incrocio"
                           pronto_R := "M_Pronto_R",
                           Pass := "Sensore_Fine_Incrocio",
                           VAI_P => "M_VAI_P",
                           VAI_R => "M_VAI_R");
END_REGION

REGION Network 6: Deviatore Pacchi
   // Istanziazione FB_Deviatore per i pacchi. Il blocco è alimentato direttamente dal sensore fisico di transito. Poiché il sensore hardware di Factory IO opera nativamente a logica inversa, il segnale viene passato all'FB tramite un contatto Normalmente Aperto.
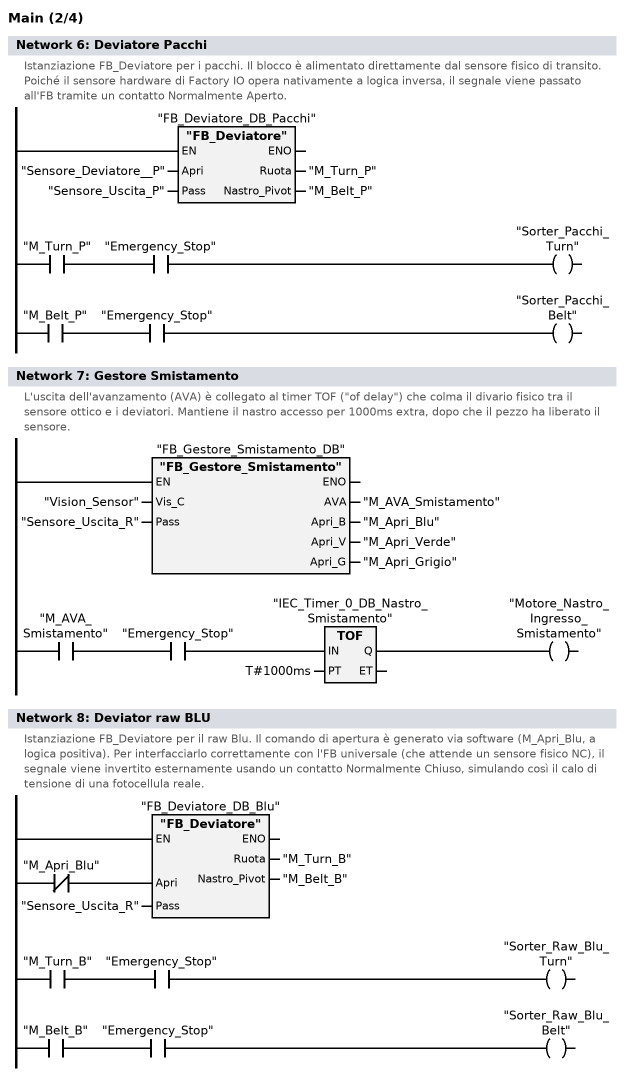
   RUNG wire#powerrail
      "FB_Deviatore_DB_Pacchi"(Apri := "Sensore_Deviatore__P", Pass := "Sensore_Uscita_P", Ruota => "M_Turn_P", Nastro_Pivot => "M_Belt_P")
   END_RUNG
   RUNG wire#powerrail
      Contact( "M_Turn_P" )
      Contact( "Emergency_Stop" )
      Coil( "Sorter_Pacchi_Turn" )
   END_RUNG
   RUNG wire#powerrail
      Contact( "M_Belt_P" )
      Contact( "Emergency_Stop" )
      Coil( "Sorter_Pacchi_Belt" )
   END_RUNG
   // the same network as SCL:
   "FB_Deviatore_DB_Pacchi"(Apri := "Sensore_Deviatore__P",   // "FB_Deviatore"
                           Pass := "Sensore_Uscita_P",
                           Ruota => "M_Turn_P",
                           Nastro_Pivot => "M_Belt_P");
   "Sorter_Pacchi_Turn" := "M_Turn_P" AND "Emergency_Stop";
   "Sorter_Pacchi_Belt" := "M_Belt_P" AND "Emergency_Stop";
END_REGION

REGION Network 7: Gestore Smistamento
   // L'uscita dell'avanzamento (AVA) è collegato al timer TOF ("of delay") che colma il divario fisico tra il sensore ottico e i deviatori. Mantiene il nastro accesso per 1000ms extra, dopo che il pezzo ha liberato il sensore.
   "FB_Gestore_Smistamento_DB"(Vis_C := "Vision_Sensor",   // "FB_Gestore_Smistamento"
                           Pass := "Sensore_Uscita_R",
                           AVA => "M_AVA_Smistamento",
                           Apri_B => "M_Apri_Blu",
                           Apri_V => "M_Apri_Verde",
                           Apri_G => "M_Apri_Grigio");
   "IEC_Timer_0_DB_Nastro_Smistamento".TOF(IN := "M_AVA_Smistamento" AND "Emergency_Stop", PT := T#1000ms);
   "Motore_Nastro_Ingresso_Smistamento" := "IEC_Timer_0_DB_Nastro_Smistamento".Q;
END_REGION

REGION Network 8: Deviator raw BLU
   // Istanziazione FB_Deviatore per il raw Blu. Il comando di apertura è generato via software (M_Apri_Blu, a logica positiva). Per interfacciarlo correttamente con l'FB universale (che attende un sensore fisico NC), il segnale viene invertito esternamente usando un contatto Normalmente Chiuso, simulando così il calo di tensione di una fotocellula reale.
   RUNG wire#powerrail
      "FB_Deviatore_DB_Blu"(Apri := wire#w1, Pass := "Sensore_Uscita_R", Ruota => "M_Turn_B", Nastro_Pivot => "M_Belt_B")
   END_RUNG
   RUNG wire#powerrail
      I_Contact( "M_Apri_Blu" )
   END_RUNG wire#w1
   RUNG wire#powerrail
      Contact( "M_Turn_B" )
      Contact( "Emergency_Stop" )
      Coil( "Sorter_Raw_Blu_Turn" )
   END_RUNG
   RUNG wire#powerrail
      Contact( "M_Belt_B" )
      Contact( "Emergency_Stop" )
      Coil( "Sorter_Raw_Blu_Belt" )
   END_RUNG
   // the same network as SCL:
   "FB_Deviatore_DB_Blu"(Apri := NOT "M_Apri_Blu",   // "FB_Deviatore"
                         Pass := "Sensore_Uscita_R",
                         Ruota => "M_Turn_B",
                         Nastro_Pivot => "M_Belt_B");
   "Sorter_Raw_Blu_Turn" := "M_Turn_B" AND "Emergency_Stop";
   "Sorter_Raw_Blu_Belt" := "M_Belt_B" AND "Emergency_Stop";
END_REGION

REGION Network 9: Deviatore raw VERDE
   // Idem a Network 8
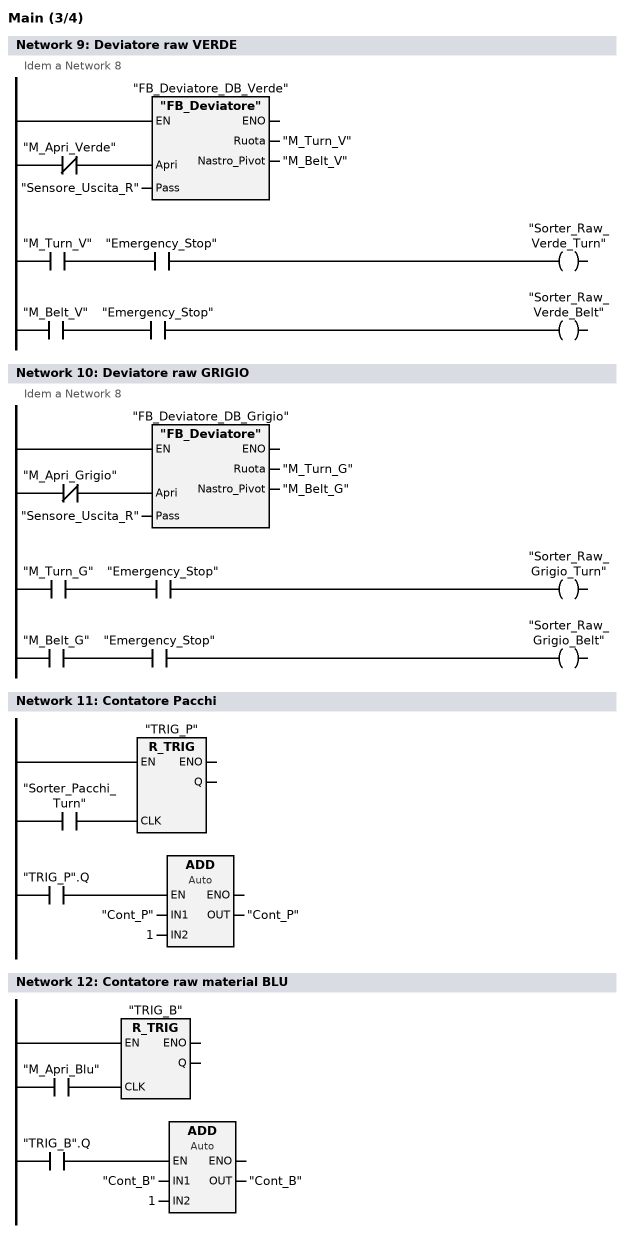
   RUNG wire#powerrail
      "FB_Deviatore_DB_Verde"(Apri := wire#w1, Pass := "Sensore_Uscita_R", Ruota => "M_Turn_V", Nastro_Pivot => "M_Belt_V")
   END_RUNG
   RUNG wire#powerrail
      I_Contact( "M_Apri_Verde" )
   END_RUNG wire#w1
   RUNG wire#powerrail
      Contact( "M_Turn_V" )
      Contact( "Emergency_Stop" )
      Coil( "Sorter_Raw_Verde_Turn" )
   END_RUNG
   RUNG wire#powerrail
      Contact( "M_Belt_V" )
      Contact( "Emergency_Stop" )
      Coil( "Sorter_Raw_Verde_Belt" )
   END_RUNG
   // the same network as SCL:
   "FB_Deviatore_DB_Verde"(Apri := NOT "M_Apri_Verde",   // "FB_Deviatore"
                           Pass := "Sensore_Uscita_R",
                           Ruota => "M_Turn_V",
                           Nastro_Pivot => "M_Belt_V");
   "Sorter_Raw_Verde_Turn" := "M_Turn_V" AND "Emergency_Stop";
   "Sorter_Raw_Verde_Belt" := "M_Belt_V" AND "Emergency_Stop";
END_REGION

REGION Network 10: Deviatore raw GRIGIO
   // Idem a Network 8
   RUNG wire#powerrail
      "FB_Deviatore_DB_Grigio"(Apri := wire#w1, Pass := "Sensore_Uscita_R", Ruota => "M_Turn_G", Nastro_Pivot => "M_Belt_G")
   END_RUNG
   RUNG wire#powerrail
      I_Contact( "M_Apri_Grigio" )
   END_RUNG wire#w1
   RUNG wire#powerrail
      Contact( "M_Turn_G" )
      Contact( "Emergency_Stop" )
      Coil( "Sorter_Raw_Grigio_Turn" )
   END_RUNG
   RUNG wire#powerrail
      Contact( "M_Belt_G" )
      Contact( "Emergency_Stop" )
      Coil( "Sorter_Raw_Grigio_Belt" )
   END_RUNG
   // the same network as SCL:
   "FB_Deviatore_DB_Grigio"(Apri := NOT "M_Apri_Grigio",   // "FB_Deviatore"
                           Pass := "Sensore_Uscita_R",
                           Ruota => "M_Turn_G",
                           Nastro_Pivot => "M_Belt_G");
   "Sorter_Raw_Grigio_Turn" := "M_Turn_G" AND "Emergency_Stop";
   "Sorter_Raw_Grigio_Belt" := "M_Belt_G" AND "Emergency_Stop";
END_REGION

REGION Network 11: Contatore Pacchi
   "TRIG_P"(CLK := "Sorter_Pacchi_Turn");   // R_TRIG
   IF "TRIG_P".Q THEN "Cont_P" := "Cont_P" + 1; END_IF;
END_REGION

REGION Network 12: Contatore raw material BLU
   "TRIG_B"(CLK := "M_Apri_Blu");   // R_TRIG
   IF "TRIG_B".Q THEN "Cont_B" := "Cont_B" + 1; END_IF;
END_REGION

REGION Network 13: Contatore raw material VERDI
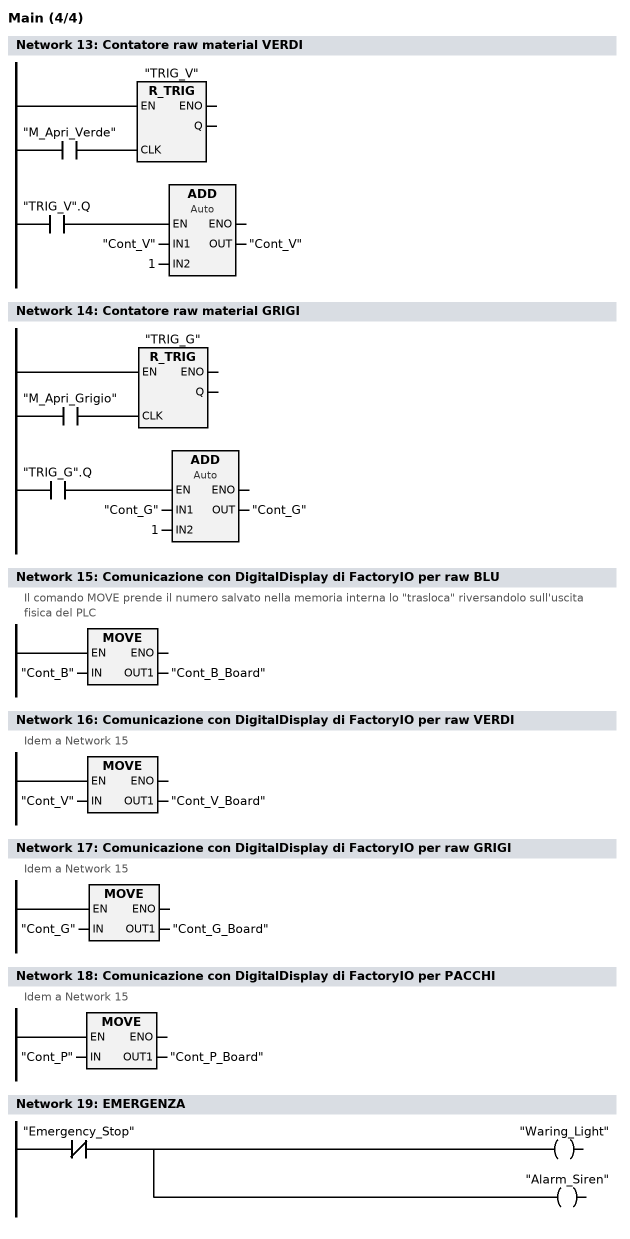
   "TRIG_V"(CLK := "M_Apri_Verde");   // R_TRIG
   IF "TRIG_V".Q THEN "Cont_V" := "Cont_V" + 1; END_IF;
END_REGION

REGION Network 14: Contatore raw material GRIGI
   "TRIG_G"(CLK := "M_Apri_Grigio");   // R_TRIG
   IF "TRIG_G".Q THEN "Cont_G" := "Cont_G" + 1; END_IF;
END_REGION

REGION Network 15: Comunicazione con DigitalDisplay di FactoryIO per raw BLU
   // Il comando MOVE prende il numero salvato nella memoria interna lo "trasloca" riversandolo sull'uscita fisica del PLC
   RUNG wire#powerrail
      Move(in := "Cont_B", out1 => "Cont_B_Board")
   END_RUNG
   // the same network as SCL:
   "Cont_B_Board" := "Cont_B";
END_REGION

REGION Network 16: Comunicazione con DigitalDisplay di FactoryIO per raw VERDI
   // Idem a Network 15
   RUNG wire#powerrail
      Move(in := "Cont_V", out1 => "Cont_V_Board")
   END_RUNG
   // the same network as SCL:
   "Cont_V_Board" := "Cont_V";
END_REGION

REGION Network 17: Comunicazione con DigitalDisplay di FactoryIO per raw GRIGI
   // Idem a Network 15
   RUNG wire#powerrail
      Move(in := "Cont_G", out1 => "Cont_G_Board")
   END_RUNG
   // the same network as SCL:
   "Cont_G_Board" := "Cont_G";
END_REGION

REGION Network 18: Comunicazione con DigitalDisplay di FactoryIO per PACCHI
   // Idem a Network 15
   RUNG wire#powerrail
      Move(in := "Cont_P", out1 => "Cont_P_Board")
   END_RUNG
   // the same network as SCL:
   "Cont_P_Board" := "Cont_P";
END_REGION

REGION Network 19: EMERGENZA
   RUNG wire#powerrail
      I_Contact( "Emergency_Stop" )
      wire#w1
      Coil( "Waring_Light" )
   END_RUNG
   RUNG wire#w1
      Coil( "Alarm_Siren" )
   END_RUNG
   // the same network as SCL:
   "Waring_Light" := NOT "Emergency_Stop";
   "Alarm_Siren" := NOT "Emergency_Stop";
END_REGION
END_ORGANIZATION_BLOCK

(* ===== HMI "HMI_RT_1" =====
system functions are stored by id; their names below are inferred from use
connection "HMI_Connection_1": ETHERNET, SMART_S7_1200_OMS
connection "HMI_Connection_2": ETHERNET, SMART_S7_1200_OMS

HMI tags "Default tag table"
   "Tag_ScreenNumber" : UInt, internal
   "Cont_B" : Int = PLC Cont_B AT %MW100, 1 s
   "Cont_V" : Int = PLC Cont_V AT %MW102, 1 s
   "Cont_G" : Int = PLC Cont_G AT %MW104, 1 s
   "Cont_P" : Int = PLC Cont_P AT %MW106, 1 s
   "Motore_Nastro_Comune" : Bool = PLC Motore_Nastro_Comune AT %Q2.0, 1 s

analog alarms
   1: 'ATTENZIONE: Smistati più di 5 raw material Blu!', class Errors, trigger "Cont_B"
   2: 'ATTENZIONE: Smistati più di 5 raw material Verdi!', class Errors, trigger "Cont_V"
   3: 'ATTENZIONE: Smistati più di 5 raw material Grigi!', class Errors, trigger "Cont_G"
   4: 'ATTENZIONE: Smistati più di 10 Pacchi!', class Errors, trigger "Cont_P"

Template "Template_1" 800x480
   Button "Exit" at 722,440 size 55x39; TextOff 'Exit'; PictureOff "ExitRuntime_KTP900_Basic_PN_TR"; PictureOn "ExitRuntime_KTP900_Basic_PN_TR"
      on Release: StopRuntime(0)
   Button "Template_Button" at 622,440 size 55x39; TextOff 'Text'
   Button "Template_Button_1" at 522,440 size 55x39; TextOff 'Text'
   Button "Template_Button_2" at 422,440 size 55x39; TextOff 'Text'
   Button "Template_Button_3" at 322,440 size 55x39; TextOff 'Text'
   Button "Template_Button_4" at 222,440 size 55x39; TextOff 'Text'
   Button "Alarms" at 122,440 size 55x39; TextOff 'Alarms'; PictureOff "AlarmDisplay_KTP900_Basic_PN_TR"; PictureOn "AlarmDisplay_KTP900_Basic_PN_TR"
      on Release: function_ef3f5d25("Alarm window_Unacknowledged", -1)
   Button "Start screen" at 22,440 size 55x39; TextOff 'Start screen'; PictureOff "NavigateHome_KTP900_Basic_PN_TR"; PictureOn "NavigateHome_KTP900_Basic_PN_TR"
      on Release: ActivateScreen("DOUBLE SORTING SYSTEM", 0)
   SymbolicIOField "Symbolic_IO_Field_Screen" at 73,7 size 620x26; TextOff '0'; TextOn '1'; TextList "TextList_ScreenNames"
      ProcessValue <- "Tag_ScreenNumber"
      on Change: ActivateScreenByNumber("Tag_ScreenNumber", 0)
   DateTimeField "HmiScreenItemData" at 695,20 size 105x20
   DateTimeField "HmiScreenItemData_1" at 695,0 size 105x20
   GraphicView "Logo" at 0,0 size 71x40; Picture "Logo of HMI_1"

screen "DOUBLE SORTING SYSTEM" 800x480, template "Template_1"
   on GenerateScreen: SetTag("Tag_ScreenNumber", 1)
   TextField "HmiScreenItemData" at 80,226 size 640x22; Text 'Text'
   Circle "Circle_1" at 307,63 size 48x48
      Appearance <- "Motore_Nastro_Comune"
   TextField "Text field_1" at 64,137 size 224x34; Text 'CONTATORI RAW'
   TextField "Text field_2" at 66,187 size 43x27; Text 'BLU'
   TextField "Text field_3" at 64,233 size 70x27; Text 'VERDE'
   TextField "Text field_4" at 62,71 size 226x34; Text 'STATO IMPIANTO'
   TextField "Text field_5" at 64,284 size 80x27; Text 'GRIGIO'
   IOField "I/O field_1" at 162,187 size 96x32; FormatPattern s999
      ProcessValue <- "Cont_B"
   IOField "I/O field_2" at 162,237 size 96x32; FormatPattern s999
      ProcessValue <- "Cont_V"
   IOField "I/O field_3" at 162,279 size 96x32; FormatPattern s999
      ProcessValue <- "Cont_G"
   TextField "Text field_6" at 419,137 size 261x34; Text 'CONTATORI PACCHI'
   TextField "Text field_7" at 422,187 size 80x27; Text 'PACCHI'
   IOField "I/O field_4" at 526,182 size 96x32; FormatPattern s999
      ProcessValue <- "Cont_P"
*)